// TwinCAT 3 PLC project SampleVision
// ProgramVersion: 3.1.4024.0
// libraries:
//   Tc2_Standard, * (Beckhoff Automation GmbH)
//   Tc2_System, * (Beckhoff Automation GmbH)
//   Tc3_Module, * (Beckhoff Automation GmbH)
//   Tc3_Vision, * (Beckhoff Automation GmbH)
// project tree:
//   DUTs/ LED1904.TcDUT
//   GVLs/ Globale_Definitionen.TcGVL, Globale_Kamera_Variablen.TcGVL
//   / PlcTask.TcTTO
//   POUs/ Camera.TcPOU, MAIN.TcPOU, MAIN_1.TcPOU
// (motion and I/O tree: see PLC project plc1)
// real-time tasks:
//   TASK PlcTask: cycle T#10ms, priority 20, ADS port 350
//   TASK PlcTask1: cycle T#10ms, priority 21, ADS port 351
//   TASK PlcTask2: cycle T#10ms, priority 22, ADS port 352

CONFIGURATION SampleVision
    RESOURCE PLC ON TwinCAT3
        TASK PlcTask(INTERVAL := T#10ms, PRIORITY := 21);
        PROGRAM MAIN WITH PlcTask : MAIN;
    END_RESOURCE
END_CONFIGURATION

// ---- DUTs/LED1904.TcDUT
TYPE LED1904 :
STRUCT
	bInput1:BOOL;
	bInput2:BOOL;
	bInput3:BOOL;
	bInput4:BOOL;
	bDiag1:BOOL;
	bDiag2:BOOL;
	bDiag3:BOOL;
	bDiag4:BOOL;
END_STRUCT
END_TYPE

// ---- GVLs/Globale_Definitionen.TcGVL
{attribute 'Tc2GvlVarNames'}
VAR_GLOBAL
	FileName: STRING := 'C:\TwinSAFE\TestErgebnisse\EL1904\TestLog_EL1904_';
	StartUp_Wait_Time: TIME := t#3s;
	ShutDown_Wait_Time : TIME := T#1S;
	Kamera_Wait_Time: TIME := T#2S;
	Prisma_Wait_Time:  TIME := T#3S;
	Seriell_Wait_Time: TIME := T#1S;
	KameraBeleuchtungFaktorWarteZeit:UINT:=8;
	Kopfzeile: STRING(255);
	TesterArray: ARRAY[0..7] OF STRING ;
	EtherCATAmsNetID: T_AmsNetId := '172.16.3.218.2.1';
	EL1904port: T_AmsPort := 1024;
	EL6900port: T_AmsPort := 1010;
	OutputWait_Time: TIME := t#5s;
	Color_Rot : DWORD := 16#000000FF;
	Color_Gruen : DWORD := 16#00007F00;
	Color_Weiss : DWORD := 16#00FFFFFF;
	Color_Visu : DWORD := 16#00FFFFFF;
	VoltagePowerContacts20Vunder : UINT := 21300; (* 0V = 0, 30V = 32767  1092 pro Volt  20V = 21845*)
	VoltagePowerContacts20Vover : UINT := 22300; (* 0V = 0, 30V = 32767  1092 pro Volt  20V = 21845*)
	VoltagePowerContacts24Vunder : UINT := 25900; (* 0V = 0, 30V = 32767  1092 pro Volt  24V = 26213*)
	VoltagePowerContacts24Vover : UINT := 26700; (* 0V = 0, 30V = 32767  1092 pro Volt  24V = 26213*)
	VoltagePowerContacts30Vunder : UINT := 32200; (* 0V = 0, 30V = 32767  1092 pro Volt  30V = 32767*)
	VoltagePowerContacts30Vover : UINT := 32767; (* 0V = 0, 30V = 32767  1092 pro Volt  30V = 32767*)
	LogFileSerialNumber: UDINT;
	Artikel : UDINT := 70931;
//	SafetyProg1: T_MaxString := 'C:\TwinSAFE\Programm\EL\Automated_EL1904\1_SafetyProgramCRC';
//	SafetyCRC1: WORD := 17617;
	SafetyProg65534: T_MaxString := 'C:\TwinSAFE\Programm\EL\Automated_EL1904\65534_SafetyProgramCRC';
	SafetyCRC65534: WORD := 65346;
END_VAR

// ---- GVLs/Globale_Kamera_Variablen.TcGVL
{attribute 'qualified_only'}
VAR_GLOBAL
	//TestVariablen
	bStopStepPrismaDetection:BOOL:=FALSE;
	bStopStepAllLedOn:BOOL:=FALSE;
	bEinrichtBetrieb:BOOL:=FALSE;
	bNextStepEinrichtbetrieb:BOOL:=FALSE;
	bPrismaOk:BOOL:=FALSE;
	bPrismaNotOK:BOOL:=FALSE;
	
	//Kamera aktiv
	bKameraAktiv:BOOL:=TRUE;
	
	//erkannte LEDs
	bLED_TermXOn		: ARRAY  [1..8] OF LED1904;
	iDetectedLED			: INT:=0;
	iStartDetectedLED		: INT:=1;
	
	// Color Simularity
	aRefColor					:	TcVnPoint3_LREAL;
	aRefColorGreen				:	TcVnPoint3_LREAL	:= [130, 230, 0];
	aRefColorRed				:	TcVnPoint3_LREAL	:= [255, 255, 255];
	aRefColorPrismError			:	TcVnPoint3_LREAL	:= [135, 150, 105];
	fVariance					:	REAL := 0.10;
	fLuminanceWeight			:	REAL := 0.1;
	
	//Threshold
	fThreshold					:	LREAL;	(* fixed threshold (unused if dynamic thresholding is selected) *)
	fMaxValue					:	LREAL;	(* maximum pixel value *)

	fThresholdGreenLed			:	LREAL:= 10 ;	(* fixed threshold (unused if dynamic thresholding is selected) *)
	fMaxValueGreenLed			:	LREAL:= 255;	(* maximum pixel value *)
	
	fThresholdRedLed			:	LREAL:= 15 ;	(* fixed threshold (unused if dynamic thresholding is selected) *)
	fMaxValueRedLed			:	LREAL:= 255;	(* maximum pixel value *)
	
	fThreshold_Prism			:	LREAL:= 185 ;	(* fixed threshold (unused if dynamic thresholding is selected) *)
	fMaxValue_Prism				:	LREAL:= 255;	(* maximum pixel value *)
	
	//Konturen zeichnen
	fAreaMin					: 	REAL:=1200;		(*Mindestfläche der zufindenden LED*)
	fAreaMax					: 	REAL:=3000;		(*Mindestfläche der zufindenden LED*)
	fHeightMin					: 	REAL:=30;		(*Mindesthöhe der zufindenden LED*)
	fHeightMax					: 	REAL:=70;		(*Maximalhöhe der zufindenden LED*)
	fWidthMax					: 	REAL:=70;		(*Maximalhöhe der zufindenden LED*)
	
	fAreaMinLED					: 	REAL:=1200;		(*Mindestfläche der zufindenden LED*)
	fAreaMaxLED					: 	REAL:=3000;		(*Mindestfläche der zufindenden LED*)
	fHeightMinLED				: 	REAL:=30;		(*Mindesthöhe der zufindenden LED*)
	fHeightMaxLED				: 	REAL:=70;		(*Maximalhöhe der zufindenden LED*)
	fWidthMaxLED				: 	REAL:=90;		(*Maximalhöhe der zufindenden LED*)
	
	fAreaMinPrisma				: 	REAL:=450;		(*Mindestfläche der zufindenden LED*)
	fAreaMaxPrisma				: 	REAL:=900;		(*Mindestfläche der zufindenden LED*)
	fHeightMinPrisma			: 	REAL:=20;		(*Mindesthöhe der zufindenden LED*)
	fHeightMaxPrisma			: 	REAL:=70;		(*Maximalhöhe der zufindenden LED*)
	fWidthMaxPrisma				: 	REAL:=70;		(*Maximalhöhe der zufindenden LED*)
	
	// Positionsgrenzen
	uiLowerPosDeviation:UINT:=10;
	uiUpperPosDeviation:UINT:=10;
	aCenterReferenceCoordinatesXY	: ARRAY  [1..8] OF TcVnPoint2_REAL;
	CenterXPosInput1:REAL:=46;
	CenterYPosInput1:REAL:=36;
	CenterXPosInput2:REAL:=119;
	CenterYPosInput2:REAL:=33;
	CenterXPosInput3:REAL:=46;
	CenterYPosInput3:REAL:=87;
	CenterXPosInput4:REAL:=120;
	CenterYPosInput4:REAL:=87;
	CenterXPosDiag1:REAL:=46;
	CenterYPosDiag1:REAL:=139;
	CenterXPosDiag2:REAL:=114;
	CenterYPosDiag2:REAL:=137;
	CenterXPosDiag3:REAL:=45;
	CenterYPosDiag3:REAL:=192;
	CenterXPosDiag4:REAL:=124;
	CenterYPosDiag4:REAL:=192;
	
	// Region of Interrest
	nXposPrisma			:	UDINT:=1514;
	nYposPrisma			:	UDINT:=892;
	nROIWidth			:	UDINT:=170;
	nROIHeight			:	UDINT:=220;

	
	// Beleuchtung EL2595
	bLedOn AT%Q* :BOOL;
	uiOutputCurrent AT%Q*:UINT;
	bLedReset AT%Q*:BOOL;
	bLedWarning AT%I*:BOOL;
	bLedError AT%I*:BOOL;	
	uiOutputCurrentEinrichtbertieb:UINT:=300;
END_VAR

// ---- POUs/MAIN.TcPOU
PROGRAM MAIN
VAR
END_VAR

END_PROGRAM

// ---- POUs/Camera.TcPOU
PROGRAM Camera
VAR
	
hr							:	HRESULT;
fbCameraControl				:	FB_VN_GevCameraControl;    //SymbolInitialization  verlinken!
	eState						:	ETcVnCameraState;
	
	ipImgIn						:	ITcVnImage;
	ipImgRoi					:   ITcVnImage;
	ipImgRotated				:   ITcVnImage;
	ipImgConvertColorSpace		: 	ITcVnImage;
	ipImgColorSimilarity		:	ITcVnImage;
	ipImgThreshold				:	ITcVnImage;
	ipImgResult					:	ITcVnImage;
	
	ipImg_Eingangsbild				:	ITcVnDisplayableImage;
	ipImg_Ausgeschnitten			:	ITcVnDisplayableImage;
	ipImg_Gedreht					:	ITcVnDisplayableImage;
	ipImg_Farbbild					:	ITcVnDisplayableImage;
	ipImg_Farbauswahl				:	ITcVnDisplayableImage;
	ipImg_Schwellwert_Farbauswahl	:	ITcVnDisplayableImage;
	ipImg_Ergebnis					:	ITcVnDisplayableImage;
	
	
	
	// Region of Interrest
	nXposTerm1			:	UDINT;
	nYposTerm1			:	UDINT;
	nROIWidth			:	UDINT;
	nROIHeight			:	UDINT;
	
	// Get Center 
	aCenterCoordinatesXY	: ARRAY  [1..8] OF TcVnPoint2_REAL;
	
	aWhite				:	TcVnVector4_LREAL	:=	[255,255,255];
	aBlack				:	TcVnVector4_LREAL	:=	[0,0,0];
	aRed				:	TcVnVector4_LREAL	:= 	[255,0,0];
	aGreen				:	TcVnVector4_LREAL	:=	[0,255,0];
	aBlue				:	TcVnVector4_LREAL	:=	[0,0,255];
	aOrange				:	TcVnVector4_LREAL	:=	[255,150,0];
END_VAR

// Position zum Zuschneiden des Prismas aus der Visu übergeben
nXposTerm1:=Globale_Kamera_Variablen.nXposPrisma;
nYposTerm1:=Globale_Kamera_Variablen.nYposPrisma;
nROIWidth:=Globale_Kamera_Variablen.nROIWidth;
nROIHeight:=Globale_Kamera_Variablen.nROIHeight;

// Kamera Kontroll Status Maschine

eState := fbCameraControl.GetState();
//eState := fbFileSource.GetState();

CASE eState OF
	
TCVN_CS_INITIAL, TCVN_CS_OPENING, TCVN_CS_OPENED, TCVN_CS_STARTACQUISITION:
	//hr := fbFileSource.StartAcquisition();
	hr := fbCameraControl.StartAcquisition();
	
TCVN_CS_ACQUIRING:
	
	//hr := fbFileSource.GetCurrentImage(ipImgIn);
	hr := fbCameraControl.GetCurrentImage(ipImgIn);
	
	IF SUCCEEDED(hr) AND ipImgIn <> 0 THEN
		
		Detect_LED(); 		(*Methoden Aufruf*)
		
		
	
		hr := F_VN_TransformIntoDisplayableImage(ipImgIn, ipImg_Eingangsbild, S_OK);
		hr := F_VN_TransformIntoDisplayableImage(ipImgRoi, ipImg_Ausgeschnitten, S_OK);
		hr := F_VN_TransformIntoDisplayableImage(ipImgRotated, ipImg_Gedreht, S_OK);
		hr := F_VN_TransformIntoDisplayableImage(ipImgConvertColorSpace, ipImg_Farbbild, S_OK);
		hr := F_VN_TransformIntoDisplayableImage(ipImgColorSimilarity, ipImg_Farbauswahl, S_OK);
		hr := F_VN_TransformIntoDisplayableImage(ipImgThreshold, ipImg_Schwellwert_Farbauswahl, S_OK);
		hr := F_VN_TransformIntoDisplayableImage(ipImgResult, ipImg_Ergebnis, S_OK);
		
	END_IF

// Freigeben der Bilder sonst kann es zum Page Fault kommen
//	F_VN_ReleaseInterface(ipImgIn);
//	F_VN_ReleaseInterface(ipImgRoi);
//	F_VN_ReleaseInterface(ipImgRotated);
//	F_VN_ReleaseInterface(ipImgConvertColorSpace);
//	F_VN_ReleaseInterface(ipImgColorSimilarity);
//	F_VN_ReleaseInterface(ipImgThreshold);
//	F_VN_ReleaseInterface(ipImgResult);

	
	Tc3_Module.FW_SafeRelease(ADR(ipImgIn));
	Tc3_Module.FW_SafeRelease(ADR(ipImgRoi));
	Tc3_Module.FW_SafeRelease(ADR(ipImgRotated));
	Tc3_Module.FW_SafeRelease(ADR(ipImgConvertColorSpace));
	Tc3_Module.FW_SafeRelease(ADR(ipImgColorSimilarity));
	Tc3_Module.FW_SafeRelease(ADR(ipImgThreshold));
	Tc3_Module.FW_SafeRelease(ADR(ipImgResult));

	
	
	
TCVN_CS_ERROR:
	//hr := fbFileSource.Reset();
	hr := fbCameraControl.Reset();
	
	END_CASE

//Positionen der Mittelpunktskoordinaten aus der Visu übernehmen
Globale_Kamera_Variablen.aCenterReferenceCoordinatesXY[1][0]:=Globale_Kamera_Variablen.CenterXPosInput1;
Globale_Kamera_Variablen.aCenterReferenceCoordinatesXY[1][1]:=Globale_Kamera_Variablen.CenterYPosInput1;
Globale_Kamera_Variablen.aCenterReferenceCoordinatesXY[2][0]:=Globale_Kamera_Variablen.CenterXPosInput2;
Globale_Kamera_Variablen.aCenterReferenceCoordinatesXY[2][1]:=Globale_Kamera_Variablen.CenterYPosInput2;
Globale_Kamera_Variablen.aCenterReferenceCoordinatesXY[3][0]:=Globale_Kamera_Variablen.CenterXPosInput3;
Globale_Kamera_Variablen.aCenterReferenceCoordinatesXY[3][1]:=Globale_Kamera_Variablen.CenterYPosInput3;
Globale_Kamera_Variablen.aCenterReferenceCoordinatesXY[4][0]:=Globale_Kamera_Variablen.CenterXPosInput4;
Globale_Kamera_Variablen.aCenterReferenceCoordinatesXY[4][1]:=Globale_Kamera_Variablen.CenterYPosInput4;
Globale_Kamera_Variablen.aCenterReferenceCoordinatesXY[5][0]:=Globale_Kamera_Variablen.CenterXPosDiag1;
Globale_Kamera_Variablen.aCenterReferenceCoordinatesXY[5][1]:=Globale_Kamera_Variablen.CenterYPosDiag1;
Globale_Kamera_Variablen.aCenterReferenceCoordinatesXY[6][0]:=Globale_Kamera_Variablen.CenterXPosDiag2;
Globale_Kamera_Variablen.aCenterReferenceCoordinatesXY[6][1]:=Globale_Kamera_Variablen.CenterYPosDiag2;
Globale_Kamera_Variablen.aCenterReferenceCoordinatesXY[7][0]:=Globale_Kamera_Variablen.CenterXPosDiag3;
Globale_Kamera_Variablen.aCenterReferenceCoordinatesXY[7][1]:=Globale_Kamera_Variablen.CenterYPosDiag3;
Globale_Kamera_Variablen.aCenterReferenceCoordinatesXY[8][0]:=Globale_Kamera_Variablen.CenterXPosDiag4;
Globale_Kamera_Variablen.aCenterReferenceCoordinatesXY[8][1]:=Globale_Kamera_Variablen.CenterYPosDiag4;



	
//Detectiere LEDs	
//Diag1 LED
	Globale_Kamera_Variablen.iStartDetectedLED:=1;
	Globale_Kamera_Variablen.bLED_TermXOn[1].bDiag1:=FALSE;
FOR Globale_Kamera_Variablen.iStartDetectedLED:=1 TO Globale_Kamera_Variablen.iDetectedLED BY 1 DO
	IF aCenterCoordinatesXY[Globale_Kamera_Variablen.iStartDetectedLED][0] > Globale_Kamera_Variablen.aCenterReferenceCoordinatesXY[5][0] - Globale_Kamera_Variablen.uiLowerPosDeviation  AND 
		aCenterCoordinatesXY[Globale_Kamera_Variablen.iStartDetectedLED][0] < Globale_Kamera_Variablen.aCenterReferenceCoordinatesXY[5][0] + Globale_Kamera_Variablen.uiUpperPosDeviation AND 
		aCenterCoordinatesXY[Globale_Kamera_Variablen.iStartDetectedLED][1] > Globale_Kamera_Variablen.aCenterReferenceCoordinatesXY[5][1] - Globale_Kamera_Variablen.uiLowerPosDeviation AND 
		aCenterCoordinatesXY[Globale_Kamera_Variablen.iStartDetectedLED][1] < Globale_Kamera_Variablen.aCenterReferenceCoordinatesXY[5][1] + Globale_Kamera_Variablen.uiUpperPosDeviation  THEN
		Globale_Kamera_Variablen.bLED_TermXOn[1].bDiag1:=TRUE;	
	END_IF
END_FOR


//Diag2 LED
	Globale_Kamera_Variablen.iStartDetectedLED:=1;
	Globale_Kamera_Variablen.bLED_TermXOn[1].bDiag2:=FALSE;
FOR Globale_Kamera_Variablen.iStartDetectedLED:=1 TO Globale_Kamera_Variablen.iDetectedLED BY 1 DO
	IF aCenterCoordinatesXY[Globale_Kamera_Variablen.iStartDetectedLED][0] > Globale_Kamera_Variablen.aCenterReferenceCoordinatesXY[6][0] - Globale_Kamera_Variablen.uiLowerPosDeviation AND 
		aCenterCoordinatesXY[Globale_Kamera_Variablen.iStartDetectedLED][0] < Globale_Kamera_Variablen.aCenterReferenceCoordinatesXY[6][0] + Globale_Kamera_Variablen.uiUpperPosDeviation AND 
	 	aCenterCoordinatesXY[Globale_Kamera_Variablen.iStartDetectedLED][1] > Globale_Kamera_Variablen.aCenterReferenceCoordinatesXY[6][1] - Globale_Kamera_Variablen.uiLowerPosDeviation AND 
		aCenterCoordinatesXY[Globale_Kamera_Variablen.iStartDetectedLED][1] < Globale_Kamera_Variablen.aCenterReferenceCoordinatesXY[6][1] + Globale_Kamera_Variablen.uiUpperPosDeviation   THEN
	Globale_Kamera_Variablen.bLED_TermXOn[1].bDiag2:=TRUE;	
	END_IF
END_FOR

//Diag3 LED
	Globale_Kamera_Variablen.iStartDetectedLED:=1;
	Globale_Kamera_Variablen.bLED_TermXOn[1].bDiag3:=FALSE;
FOR Globale_Kamera_Variablen.iStartDetectedLED:=1 TO Globale_Kamera_Variablen.iDetectedLED BY 1 DO
	IF aCenterCoordinatesXY[Globale_Kamera_Variablen.iStartDetectedLED][0] >  Globale_Kamera_Variablen.aCenterReferenceCoordinatesXY[7][0] - Globale_Kamera_Variablen.uiLowerPosDeviation AND 
		aCenterCoordinatesXY[Globale_Kamera_Variablen.iStartDetectedLED][0] < Globale_Kamera_Variablen.aCenterReferenceCoordinatesXY[7][0] + Globale_Kamera_Variablen.uiUpperPosDeviation AND
		aCenterCoordinatesXY[Globale_Kamera_Variablen.iStartDetectedLED][1] > Globale_Kamera_Variablen.aCenterReferenceCoordinatesXY[7][1] - Globale_Kamera_Variablen.uiLowerPosDeviation AND
		aCenterCoordinatesXY[Globale_Kamera_Variablen.iStartDetectedLED][1] < Globale_Kamera_Variablen.aCenterReferenceCoordinatesXY[7][1] + Globale_Kamera_Variablen.uiUpperPosDeviation   THEN
		Globale_Kamera_Variablen.bLED_TermXOn[1].bDiag3:=TRUE;	
	END_IF
END_FOR


//Diag4 LED
	Globale_Kamera_Variablen.iStartDetectedLED:=1;
	Globale_Kamera_Variablen.bLED_TermXOn[1].bDiag4:=FALSE;
FOR Globale_Kamera_Variablen.iStartDetectedLED:=1 TO Globale_Kamera_Variablen.iDetectedLED BY 1 DO
	IF aCenterCoordinatesXY[Globale_Kamera_Variablen.iStartDetectedLED][0] > Globale_Kamera_Variablen.aCenterReferenceCoordinatesXY[8][0] - Globale_Kamera_Variablen.uiLowerPosDeviation AND 
	aCenterCoordinatesXY[Globale_Kamera_Variablen.iStartDetectedLED][0] < Globale_Kamera_Variablen.aCenterReferenceCoordinatesXY[8][0] + Globale_Kamera_Variablen.uiUpperPosDeviation 	AND 
	aCenterCoordinatesXY[Globale_Kamera_Variablen.iStartDetectedLED][1] > Globale_Kamera_Variablen.aCenterReferenceCoordinatesXY[8][1] - Globale_Kamera_Variablen.uiLowerPosDeviation 	AND 
	aCenterCoordinatesXY[Globale_Kamera_Variablen.iStartDetectedLED][1] < Globale_Kamera_Variablen.aCenterReferenceCoordinatesXY[8][1] + Globale_Kamera_Variablen.uiUpperPosDeviation   THEN
	Globale_Kamera_Variablen.bLED_TermXOn[1].bDiag4:=TRUE;	
	END_IF
END_FOR

//Input1 LED
Globale_Kamera_Variablen.iStartDetectedLED:=1;
Globale_Kamera_Variablen.bLED_TermXOn[1].bInput1:=FALSE;
FOR Globale_Kamera_Variablen.iStartDetectedLED:=1 TO Globale_Kamera_Variablen.iDetectedLED BY 1 DO
	IF aCenterCoordinatesXY[Globale_Kamera_Variablen.iStartDetectedLED][0] > Globale_Kamera_Variablen.aCenterReferenceCoordinatesXY[1][0] - Globale_Kamera_Variablen.uiLowerPosDeviation AND 
	aCenterCoordinatesXY[Globale_Kamera_Variablen.iStartDetectedLED][0] < Globale_Kamera_Variablen.aCenterReferenceCoordinatesXY[1][0] + Globale_Kamera_Variablen.uiUpperPosDeviation AND 
	aCenterCoordinatesXY[Globale_Kamera_Variablen.iStartDetectedLED][1] > Globale_Kamera_Variablen.aCenterReferenceCoordinatesXY[1][1] - Globale_Kamera_Variablen.uiLowerPosDeviation AND 
	aCenterCoordinatesXY[Globale_Kamera_Variablen.iStartDetectedLED][1] < Globale_Kamera_Variablen.aCenterReferenceCoordinatesXY[1][1] + Globale_Kamera_Variablen.uiUpperPosDeviation   THEN
	Globale_Kamera_Variablen.bLED_TermXOn[1].bInput1:=TRUE;	
	END_IF
END_FOR


//Input2 LED
Globale_Kamera_Variablen.iStartDetectedLED:=1;
Globale_Kamera_Variablen.bLED_TermXOn[1].bInput2:=FALSE;
FOR Globale_Kamera_Variablen.iStartDetectedLED:=1 TO Globale_Kamera_Variablen.iDetectedLED BY 1 DO
	IF aCenterCoordinatesXY[Globale_Kamera_Variablen.iStartDetectedLED][0] > Globale_Kamera_Variablen.aCenterReferenceCoordinatesXY[2][0] - Globale_Kamera_Variablen.uiLowerPosDeviation AND 
	aCenterCoordinatesXY[Globale_Kamera_Variablen.iStartDetectedLED][0] <  Globale_Kamera_Variablen.aCenterReferenceCoordinatesXY[2][0] + Globale_Kamera_Variablen.uiUpperPosDeviation AND 
	aCenterCoordinatesXY[Globale_Kamera_Variablen.iStartDetectedLED][1] > Globale_Kamera_Variablen.aCenterReferenceCoordinatesXY[2][1] - Globale_Kamera_Variablen.uiLowerPosDeviation AND 
	aCenterCoordinatesXY[Globale_Kamera_Variablen.iStartDetectedLED][1] < Globale_Kamera_Variablen.aCenterReferenceCoordinatesXY[2][1] + Globale_Kamera_Variablen.uiUpperPosDeviation   THEN
	Globale_Kamera_Variablen.bLED_TermXOn[1].bInput2:=TRUE;	
	END_IF
END_FOR


//Input3 LED
Globale_Kamera_Variablen.iStartDetectedLED:=1;
Globale_Kamera_Variablen.bLED_TermXOn[1].bInput3:=FALSE;
FOR Globale_Kamera_Variablen.iStartDetectedLED:=1 TO Globale_Kamera_Variablen.iDetectedLED BY 1 DO
	IF aCenterCoordinatesXY[Globale_Kamera_Variablen.iStartDetectedLED][0] > Globale_Kamera_Variablen.aCenterReferenceCoordinatesXY[3][0] - Globale_Kamera_Variablen.uiLowerPosDeviation AND 
	aCenterCoordinatesXY[Globale_Kamera_Variablen.iStartDetectedLED][0] < Globale_Kamera_Variablen.aCenterReferenceCoordinatesXY[3][0] + Globale_Kamera_Variablen.uiUpperPosDeviation AND 
	aCenterCoordinatesXY[Globale_Kamera_Variablen.iStartDetectedLED][1] > Globale_Kamera_Variablen.aCenterReferenceCoordinatesXY[3][1] - Globale_Kamera_Variablen.uiLowerPosDeviation AND 
	aCenterCoordinatesXY[Globale_Kamera_Variablen.iStartDetectedLED][1] < Globale_Kamera_Variablen.aCenterReferenceCoordinatesXY[3][1] + Globale_Kamera_Variablen.uiUpperPosDeviation   THEN
	Globale_Kamera_Variablen.bLED_TermXOn[1].bInput3:=TRUE;	
	END_IF
END_FOR


//Input4 LED
Globale_Kamera_Variablen.iStartDetectedLED:=1;
Globale_Kamera_Variablen.bLED_TermXOn[1].bInput4:=FALSE;
FOR Globale_Kamera_Variablen.iStartDetectedLED:=1 TO Globale_Kamera_Variablen.iDetectedLED BY 1 DO
	IF aCenterCoordinatesXY[Globale_Kamera_Variablen.iStartDetectedLED][0] > Globale_Kamera_Variablen.aCenterReferenceCoordinatesXY[4][0] - Globale_Kamera_Variablen.uiLowerPosDeviation AND 
	aCenterCoordinatesXY[Globale_Kamera_Variablen.iStartDetectedLED][0] < Globale_Kamera_Variablen.aCenterReferenceCoordinatesXY[4][0] + Globale_Kamera_Variablen.uiUpperPosDeviation AND 
	aCenterCoordinatesXY[Globale_Kamera_Variablen.iStartDetectedLED][1] > Globale_Kamera_Variablen.aCenterReferenceCoordinatesXY[4][1] - Globale_Kamera_Variablen.uiLowerPosDeviation AND 
	aCenterCoordinatesXY[Globale_Kamera_Variablen.iStartDetectedLED][1] < Globale_Kamera_Variablen.aCenterReferenceCoordinatesXY[4][1] + Globale_Kamera_Variablen.uiUpperPosDeviation   THEN
	Globale_Kamera_Variablen.bLED_TermXOn[1].bInput4:=TRUE;
	END_IF
END_FOR


// Center Rücksetzen, damit neuer durchlauf starten kann.
IF Globale_Kamera_Variablen.iStartDetectedLED = 0 THEN
	aCenterCoordinatesXY[1][0]:=0;
	aCenterCoordinatesXY[1][1]:=0;
	aCenterCoordinatesXY[2][0]:=0;
	aCenterCoordinatesXY[2][1]:=0;
	aCenterCoordinatesXY[3][0]:=0;
	aCenterCoordinatesXY[3][1]:=0;
	aCenterCoordinatesXY[4][0]:=0;
	aCenterCoordinatesXY[4][1]:=0;
	aCenterCoordinatesXY[5][0]:=0;
	aCenterCoordinatesXY[5][1]:=0;
	aCenterCoordinatesXY[6][0]:=0;
	aCenterCoordinatesXY[6][1]:=0;
	aCenterCoordinatesXY[7][0]:=0;
	aCenterCoordinatesXY[7][1]:=0;
	aCenterCoordinatesXY[8][0]:=0;
	aCenterCoordinatesXY[8][1]:=0;
END_IF

IF Globale_Kamera_Variablen.iStartDetectedLED = 1 THEN
	aCenterCoordinatesXY[2][0]:=0;
	aCenterCoordinatesXY[2][1]:=0;
	aCenterCoordinatesXY[3][0]:=0;
	aCenterCoordinatesXY[3][1]:=0;
	aCenterCoordinatesXY[4][0]:=0;
	aCenterCoordinatesXY[4][1]:=0;
	aCenterCoordinatesXY[5][0]:=0;
	aCenterCoordinatesXY[5][1]:=0;
	aCenterCoordinatesXY[6][0]:=0;
	aCenterCoordinatesXY[6][1]:=0;
	aCenterCoordinatesXY[7][0]:=0;
	aCenterCoordinatesXY[7][1]:=0;
	aCenterCoordinatesXY[8][0]:=0;
	aCenterCoordinatesXY[8][1]:=0;
END_IF

IF Globale_Kamera_Variablen.iStartDetectedLED = 2 THEN
	aCenterCoordinatesXY[3][0]:=0;
	aCenterCoordinatesXY[3][1]:=0;
	aCenterCoordinatesXY[4][0]:=0;
	aCenterCoordinatesXY[4][1]:=0;
	aCenterCoordinatesXY[5][0]:=0;
	aCenterCoordinatesXY[5][1]:=0;
	aCenterCoordinatesXY[6][0]:=0;
	aCenterCoordinatesXY[6][1]:=0;
	aCenterCoordinatesXY[7][0]:=0;
	aCenterCoordinatesXY[7][1]:=0;
	aCenterCoordinatesXY[8][0]:=0;
	aCenterCoordinatesXY[8][1]:=0;
END_IF

IF Globale_Kamera_Variablen.iStartDetectedLED = 3 THEN
	aCenterCoordinatesXY[4][0]:=0;
	aCenterCoordinatesXY[4][1]:=0;
	aCenterCoordinatesXY[5][0]:=0;
	aCenterCoordinatesXY[5][1]:=0;
	aCenterCoordinatesXY[6][0]:=0;
	aCenterCoordinatesXY[6][1]:=0;
	aCenterCoordinatesXY[7][0]:=0;
	aCenterCoordinatesXY[7][1]:=0;
	aCenterCoordinatesXY[8][0]:=0;
	aCenterCoordinatesXY[8][1]:=0;
END_IF

IF Globale_Kamera_Variablen.iStartDetectedLED = 4 THEN
	aCenterCoordinatesXY[5][0]:=0;
	aCenterCoordinatesXY[5][1]:=0;
	aCenterCoordinatesXY[6][0]:=0;
	aCenterCoordinatesXY[6][1]:=0;
	aCenterCoordinatesXY[7][0]:=0;
	aCenterCoordinatesXY[7][1]:=0;
	aCenterCoordinatesXY[8][0]:=0;
	aCenterCoordinatesXY[8][1]:=0;
END_IF

IF Globale_Kamera_Variablen.iStartDetectedLED = 5 THEN
	aCenterCoordinatesXY[6][0]:=0;
	aCenterCoordinatesXY[6][1]:=0;
	aCenterCoordinatesXY[7][0]:=0;
	aCenterCoordinatesXY[7][1]:=0;
	aCenterCoordinatesXY[8][0]:=0;
	aCenterCoordinatesXY[8][1]:=0;
END_IF

IF Globale_Kamera_Variablen.iStartDetectedLED = 6 THEN
	aCenterCoordinatesXY[7][0]:=0;
	aCenterCoordinatesXY[7][1]:=0;
	aCenterCoordinatesXY[8][0]:=0;
	aCenterCoordinatesXY[8][1]:=0;
END_IF

IF Globale_Kamera_Variablen.iStartDetectedLED = 7 THEN
	aCenterCoordinatesXY[8][0]:=0;
	aCenterCoordinatesXY[8][1]:=0;
END_IF

METHOD Detect_LED 
VAR
	ipImgWork			:	ITcVnImage;
	
	ipContours			:	ITcVnContainer;
	ipContour			:	ITcVnContainer;
	ipForwardIterator	:	ITcVnForwardIterator;
	aContourOffset		:	TcVnPoint;
	
	fArea				:	LREAL;
	stRect				:	TcVnRotatedRectangle;
	
	
END_VAR

//	Region of Interrest
hr := F_VN_CopyImage(ipImgIn, ipImgRoi, hr);
hr:= F_VN_SetRoi( nXposTerm1, nYposTerm1, nROIWidth, nROIHeight,ipImgRoi ,hr);

// Rotate Image
hr:=F_VN_RotateImage(ipImgRoi,ipImgRotated,TCVN_RA_180_DEG,hr);
hr := F_VN_CopyImage(ipImgRotated, ipImgRotated, hr);

// Color Space
hr := F_VN_ConvertColorSpace(ipImgRotated (*ipImgRoi*)(*ipImgIn*), ipImgWork, ETcVNColorSpaceTransform.TCVN_CST_BAYER_GR_TO_BGR , hr); //TCVN_CST_BAYER_GR_TO_RGB TCVN_CST_BAYER_BG_TO_RGB Liegt daran wie das Bild abgeschnitten wurde
hr := F_VN_CopyImage(ipImgWork, ipImgConvertColorSpace, hr);

//Color Simularity
//hr := F_VN_ComputeReferenceColorSimilarityExp_TcVnVector3_LREAL(ipImgWork, ipImgWork, Globale_Kamera_variablen.aRefColor, Globale_Kamera_Variablen.fVariance, Globale_Kamera_Variablen.fLuminanceWeight, hr);
hr := F_VN_ReferenceColorSimilarityExp_TcVnVector3_LREAL(ipImgWork, ipImgWork, Globale_Kamera_variablen.aRefColor, Globale_Kamera_Variablen.fVariance, Globale_Kamera_Variablen.fLuminanceWeight, hr);
hr := F_VN_CopyImage(ipImgWork, ipImgColorSimilarity, hr);

//Threshold
//hr := F_VN_ApplyThreshold(ipImgWork, ipImgWork, Globale_Kamera_Variablen.fThreshold, Globale_Kamera_Variablen.fMaxValue, ETcVnThresholdType.TCVN_TT_BINARY, hr);
hr := Tc3_Vision.F_VN_Threshold(ipImgWork, ipImgWork, Globale_Kamera_Variablen.fThreshold, Globale_Kamera_Variablen.fMaxValue, ETcVnThresholdType.TCVN_TT_BINARY, hr);
hr := F_VN_CopyImage(ipImgWork, ipImgThreshold, hr);


// Contours
hr := F_VN_FindContoursExp(ipImgWork, ipContours, ETcVnContourRetrievalMode.TCVN_CRM_CONNECTED_COMPONENTS, ETcVnContourApproximationMethod.TCVN_CAM_SIMPLE, aContourOffset,hr);



IF SUCCEEDED(hr) AND ipContours <> 0 THEN
	hr := F_VN_GetForwardIterator(ipContours, ipForwardIterator, hr);
	
	// Create an Image to display the results
	hr := F_VN_ConvertColorSpace(ipImgRotated(*ipImgRoi*) (*ipImgIn*), ipImgWork, ETcVNColorSpaceTransform.TCVN_CST_BAYER_GR_TO_BGR, hr);
	
	Globale_Kamera_Variablen.iDetectedLED:=0;
	
	WHILE SUCCEEDED(hr) AND ipForwardIterator.CheckIfEnd() = S_FALSE DO
		
		hr := F_VN_GetContainer(ipForwardIterator, ipContour, hr);
		hr := F_VN_IncrementIterator(ipForwardIterator, hr);
		

		// Finding Criteria to Filter the Contours
		//============================================
		
		// (2) Area and Rectangle Shape		
		//hr := F_VN_EstimateContourArea(ipContour, fArea, hr);
		hr := Tc3_Vision.F_VN_ContourArea(ipContour, fArea, hr);
		IF fArea > Globale_Kamera_Variablen.fAreaMin THEN 
			
			//hr := F_VN_DetermineEnclosingRectangle(ipContour, stRect, hr);
			hr := Tc3_Vision.F_VN_EnclosingRectangle(ipContour, stRect, hr);
			
			Globale_Kamera_Variablen.iDetectedLED:=Globale_Kamera_Variablen.iDetectedLED+1;// Falls Bild noch nicht zugeschnitten eventuell auskommentieren wegen Exception
	 
			aCenterCoordinatesXY[Globale_Kamera_Variablen.iDetectedLED]:=stRect.aCenter; // Falls Bild noch nicht zugeschnitten eventuell auskommentieren wegen Exception

			
			// Prüfen ob "Quadratisch" 									
			IF stRect.stSize.fHeight > Globale_Kamera_Variablen.fHeightMin AND stRect.stSize.fHeight < Globale_Kamera_Variablen.fHeightMax AND stRect.stSize.fWidth < Globale_Kamera_Variablen.fWidthMax THEN 
				hr := F_VN_DrawContours(ipContour, -1, ipImgWork, aGreen, 2, hr);				
			ELSIF fArea > Globale_Kamera_Variablen.fAreaMax THEN
				hr := F_VN_DrawContours(ipContour, -1, ipImgWork, aOrange, 2, hr);
			ELSE
				hr := F_VN_DrawContours(ipContour, -1, ipImgWork, aRed, 2, hr);
			END_IF
			
		END_IF
					
		//F_VN_ReleaseInterface(ipContour);
		Tc3_Module.FW_SafeRelease(ADR(ipContour));
	END_WHILE

END_IF



hr := F_VN_CopyImage(ipImgWork, ipImgResult, hr);


// Release all Interface Pointer
//F_VN_ReleaseInterface(ipContours);
//F_VN_ReleaseInterface(ipForwardIterator);
//F_VN_ReleaseInterface(ipImgWork);
Tc3_Module.FW_SafeRelease(ADR(ipContours));
Tc3_Module.FW_SafeRelease(ADR(ipForwardIterator));
Tc3_Module.FW_SafeRelease(ADR(ipImgWork));
END_METHOD

END_PROGRAM

// ---- POUs/MAIN_1.TcPOU
PROGRAM MAIN_1
VAR
END_VAR


Camera();

END_PROGRAM
